FUNCTION_BLOCK App1_ProdRateandPressure (* Composite Function Block Type *)
  (* Standard: 61499-2 *)
  (* Version 0.0, 2018-11-06, 4DIAC-IDE, 4DIAC-Consortium *)
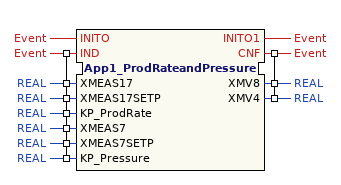
  EVENT_INPUT
    INITO; (* Initialization Request *)
    IND WITH XMEAS17, XMEAS17SETP, XMEAS7, XMEAS7SETP, KP_ProdRate, KP_Pressure; (* Normal Execution Request *)
  END_EVENT
  EVENT_OUTPUT
    INITO1; (* Initialization Confirm *)
    CNF WITH XMV8, XMV4; (* Execution Confirmation *)
  END_EVENT
  VAR_INPUT
    XMEAS17 : REAL;
    XMEAS17SETP : REAL;
    KP_ProdRate : REAL;
    XMEAS7 : REAL;
    XMEAS7SETP : REAL;
    KP_Pressure : REAL;
  END_VAR
  VAR_OUTPUT
    XMV8 : REAL;
    XMV4 : REAL;
  END_VAR
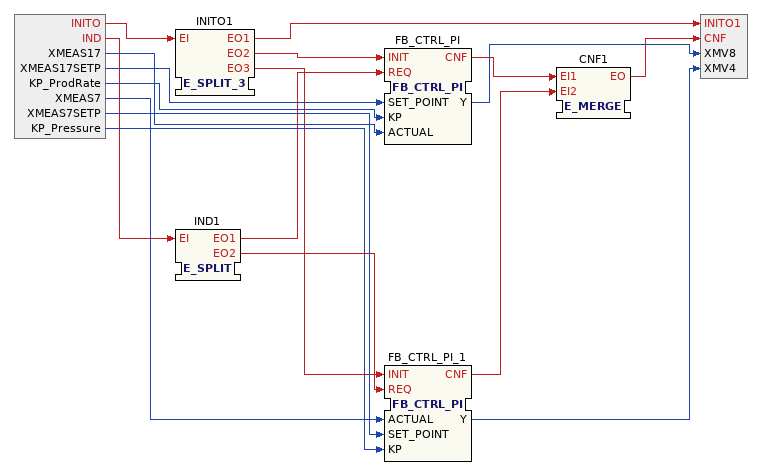
  FBS
    FB_CTRL_PI : FB_CTRL_PI;
    FB_CTRL_PI_1 : FB_CTRL_PI;
    INITO1 : E_SPLIT_3;
    IND1 : E_SPLIT;
    CNF1 : E_MERGE;
  END_FBS
  EVENT_CONNECTIONS
    CNF1.EO TO CNF;
    FB_CTRL_PI.CNF TO CNF1.EI1;
    FB_CTRL_PI_1.CNF TO CNF1.EI2;
    INITO1.EO1 TO INITO1;
    INITO1.EO2 TO FB_CTRL_PI.INIT;
    INITO1.EO3 TO FB_CTRL_PI_1.INIT;
    IND1.EO1 TO FB_CTRL_PI.REQ;
    IND1.EO2 TO FB_CTRL_PI_1.REQ;
    INITO TO INITO1.EI;
    IND TO IND1.EI;
  END_CONNECTIONS
  DATA_CONNECTIONS
    XMEAS17SETP TO FB_CTRL_PI.SET_POINT;
    XMEAS7 TO FB_CTRL_PI_1.ACTUAL;
    XMEAS7SETP TO FB_CTRL_PI_1.SET_POINT;
    FB_CTRL_PI.Y TO XMV8;
    FB_CTRL_PI_1.Y TO XMV4;
    KP_ProdRate TO FB_CTRL_PI.KP;
    KP_Pressure TO FB_CTRL_PI_1.KP;
    XMEAS17 TO FB_CTRL_PI.ACTUAL;
  END_CONNECTIONS
END_FUNCTION_BLOCK
